// TIA Portal project "Ejercicio2" (V15.1)

(* hardware
DEVICE "S7-1200 station_2"  S7-1200 Station
   slot 0: "Rack_0"  S7-1200 Rack  Rack  V1.0
   slot 1: "PLC_0"  CPU 1215C AC/DC/Rly  6ES7 215-1BG40-0XB0  V4.2
DEVICE "HMI_1"  KTP700 Basic PN Portrait
   slot 0: "HMI_1"  KTP700 Basic PN Portrait  6AV2 123-2GB03-0AX0  15.1.0.0
   slot 1: "HMI_RT_1"  KTP700 Basic PN Portrait  6AV2 123-2GB03-0AX0  15.1.0.0
   slot 5: "HMI_1.IE_CP_1"  PROFINET Interface  15.0.1.0
      slot 1: "Interfaz PROFINET_1"  PROFINET Interface
         slot 1: "Port_1"  Port
*)

// ===== PLC "PLC_0"  CPU 1215C AC/DC/Rly =====

VAR_GLOBAL   // PLC tag table "Tabla de variables estándar"
   "Zona 1" AT %M0.0 : Bool;   // Entrada delantera, sala de estar, cocina y dormitorio 3
   "Zona 2" AT %M0.1 : Bool;   // Dormitorio 1, dormitorio 2, baño y entrada trasera
   "Alarma ON/OFF" AT %M0.2 : Bool;   // Activa o desactiva el sistema de alarma.
   "Alarma manual" AT %M0.3 : Bool;   // Permite activar manualmente la sirena de alarma
   "LED sistema de alarma" AT %M10.0 : Bool;   // Estará encendido si está activado y parpadeante si está desactivado, estando abiertas la zona 1 o la zona 2
   "Sirena de alarma" AT %M10.1 : Bool;   // Dispara la sirena de alarma
   "Señal de alerta baja" AT %M10.2 : Bool;   // Activa una señal de alerta baja que indica que la alarma se disparará al cabo de un número predeterminado de segundos
   "Activar relé" AT %M10.3 : Bool;   // Activa un relé de interface externo (p.ej. para arrancar una marcación automática).
   "Estado Alarma" AT %M1.0 : Bool;   // Usaremos esta variable para detectar cuando el temporizador de 90 segundos haya pasado
   "Estado Sirena" AT %M1.1 : Bool;   // Usaremos esta variable para detectar si alguna zona esta abierta o no
END_VAR

// folder: System blocks/Program resources

DATA_BLOCK "Temporizador 90s"   // DB1
{ S7_Optimized_Access := 'TRUE' }
AUTHOR : Simatic
FAMILY : IEC
NAME : IEC_TMR
VERSION : 1.0
// stored: InstanceOfName IEC_TIMER
"IEC_TIMER"
BEGIN
END_DATA_BLOCK

DATA_BLOCK "Temporizador notificador 60s"   // DB3
{ S7_Optimized_Access := 'TRUE' }
AUTHOR : Simatic
FAMILY : IEC
NAME : IEC_TMR
VERSION : 1.0
// stored: InstanceOfName IEC_TIMER
"IEC_TIMER"
BEGIN
END_DATA_BLOCK

// folder: (top level)

ORGANIZATION_BLOCK "Main"   // OB1, LAD, ProgramCycle
TITLE = "Main Program Sweep (Cycle)"
{ S7_Optimized_Access := 'TRUE' }
VERSION : 0.1
   VAR_INPUT
      Initial_Call : Bool;   // Initial call of this OB
      Remanence : Bool;   // =True, if remanent data are available
   END_VAR
   VAR_TEMP   // added for the SCL form of the ladder/FBD networks
      _w1 : Bool;
   END_VAR
BEGIN

REGION Network 1: Estará encendido si está activado y parpadeante si está desactivado, estando abiertas la zona 1 o la zona 2
   // Si el sistema no está activado, el LED (M10.0) parpadea al estar abiertas la zona 1 (%M0.0) o 2 (%M0.1).
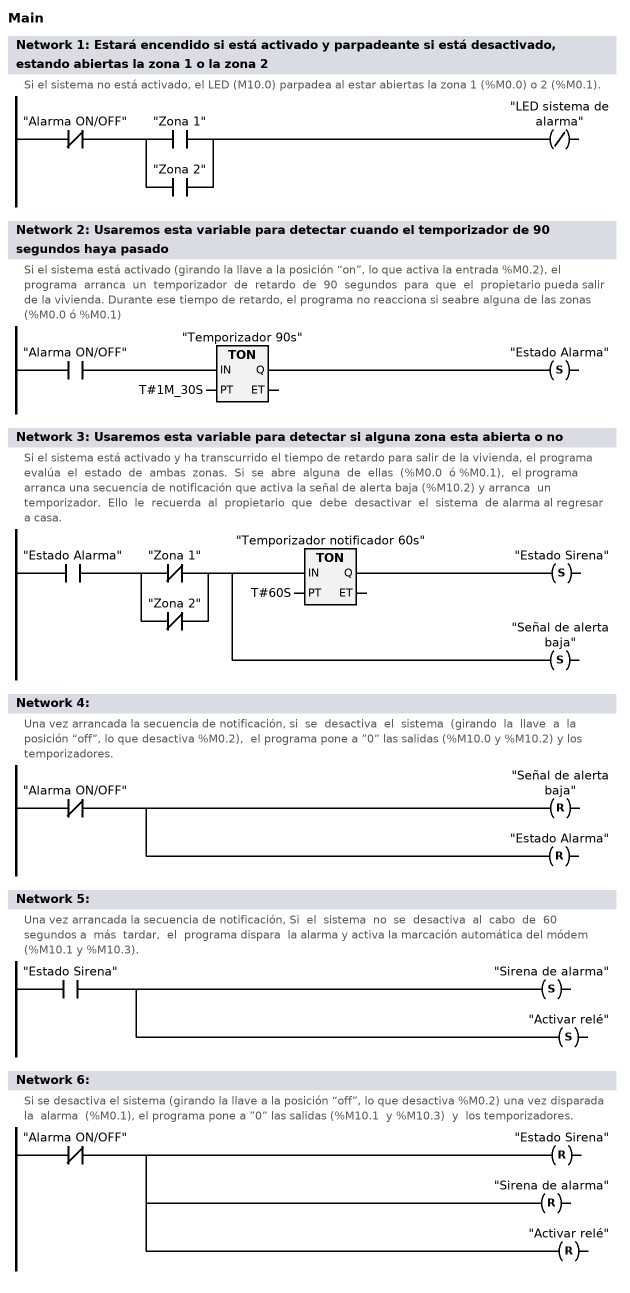
   RUNG wire#powerrail
      I_Contact( "Alarma ON/OFF" )
      wire#w1
      Contact( "Zona 1" )
      wire#w2
      I_Coil( "LED sistema de alarma" )
   END_RUNG
   RUNG wire#w1
      Contact( "Zona 2" )
   END_RUNG wire#w2
   // the same network as SCL:
   "LED sistema de alarma" := NOT (NOT "Alarma ON/OFF" AND ("Zona 1" OR "Zona 2"));
END_REGION

REGION Network 2: Usaremos esta variable para detectar cuando el temporizador de 90 segundos haya pasado
   // Si el sistema está activado (girando la llave a la posición “on”, lo que activa la entrada %M0.2), el  programa  arranca  un  temporizador  de  retardo  de  90  segundos  para  que  el  propietario pueda salir de la vivienda. Durante ese tiempo de retardo, el programa no reacciona si seabre alguna de las zonas (%M0.0 ó %M0.1)
   "Temporizador 90s".TON(IN := "Alarma ON/OFF", PT := T#1M_30S);
   IF "Temporizador 90s".Q THEN "Estado Alarma" := TRUE; END_IF;
END_REGION

REGION Network 3: Usaremos esta variable para detectar si alguna zona esta abierta o no
   // Si el sistema está activado y ha transcurrido el tiempo de retardo para salir de la vivienda, el programa  evalúa  el  estado  de  ambas  zonas.  Si  se  abre  alguna  de  ellas  (%M0.0  ó %M0.1),  el programa arranca una secuencia de notificación que activa la señal de alerta baja (%M10.2) y arranca  un  temporizador.  Ello  le  recuerda  al  propietario  que  debe  desactivar  el  sistema  de alarma al regresar a casa.
   #_w1 := "Estado Alarma" AND (NOT "Zona 1" OR NOT "Zona 2");
   "Temporizador notificador 60s".TON(IN := #_w1, PT := T#60S);
   IF "Temporizador notificador 60s".Q THEN "Estado Sirena" := TRUE; END_IF;
   IF #_w1 THEN "Señal de alerta baja" := TRUE; END_IF;
END_REGION

REGION Network 4
   // Una vez arrancada la secuencia de notificación, si  se  desactiva  el  sistema  (girando  la  llave  a  la  posición “off”, lo que desactiva %M0.2),  el programa pone a ”0” las salidas (%M10.0 y %M10.2) y los temporizadores.
   RUNG wire#powerrail
      I_Contact( "Alarma ON/OFF" )
      wire#w1
      R_Coil( "Señal de alerta baja" )
   END_RUNG
   RUNG wire#w1
      R_Coil( "Estado Alarma" )
   END_RUNG
   // the same network as SCL:
   IF NOT "Alarma ON/OFF" THEN
       "Señal de alerta baja" := FALSE;
       "Estado Alarma" := FALSE;
   END_IF;
END_REGION

REGION Network 5
   // Una vez arrancada la secuencia de notificación, Si  el  sistema  no  se  desactiva  al  cabo  de  60  segundos a  más  tardar,  el  programa dispara  la alarma y activa la marcación automática del módem (%M10.1 y %M10.3).
   RUNG wire#powerrail
      Contact( "Estado Sirena" )
      wire#w1
      S_Coil( "Sirena de alarma" )
   END_RUNG
   RUNG wire#w1
      S_Coil( "Activar relé" )
   END_RUNG
   // the same network as SCL:
   IF "Estado Sirena" THEN
       "Sirena de alarma" := TRUE;
       "Activar relé" := TRUE;
   END_IF;
END_REGION

REGION Network 6
   // Si se desactiva el sistema (girando la llave a la posición “off”, lo que desactiva %M0.2) una vez disparada  la  alarma  (%M0.1), el programa pone a ”0” las salidas (%M10.1  y %M10.3)  y  los temporizadores.
   RUNG wire#powerrail
      I_Contact( "Alarma ON/OFF" )
      wire#w1
      R_Coil( "Estado Sirena" )
   END_RUNG
   RUNG wire#w1
      R_Coil( "Sirena de alarma" )
   END_RUNG
   RUNG wire#w1
      R_Coil( "Activar relé" )
   END_RUNG
   // the same network as SCL:
   IF NOT "Alarma ON/OFF" THEN
       "Estado Sirena" := FALSE;
       "Sirena de alarma" := FALSE;
       "Activar relé" := FALSE;
   END_IF;
END_REGION
END_ORGANIZATION_BLOCK

(* ===== HMI "HMI_RT_1" =====
system functions are stored by id; their names below are inferred from use
connection "HMI_Conexión_1": ETHERNET, SMART_S7_1200_OMS

HMI tags "Tabla de variables estándar"
   "Número_imagen_variable" : UInt, internal
   "Alarma ON/OFF" : Bool = PLC "Alarma ON/OFF" AT %M0.2, 1 s
   "LED sistema de alarma" : Bool = PLC "LED sistema de alarma" AT %M10.0, 1 s
   "Señal de alerta baja" : Bool = PLC "Señal de alerta baja" AT %M10.2, 1 s
   "Sirena de alarma" : Bool = PLC "Sirena de alarma" AT %M10.1, 1 s
   "Activar relé" : Bool = PLC "Activar relé" AT %M10.3, 1 s

text list "Nombre_imagen_lista_texto": 1 'Imagen raíz'

Template "Plantilla_1" 480x800
   Button "Template_Button" at 428,727 size 50x71; TextOff 'Text'
   Button "Template_Button_1" at 375,727 size 50x71; TextOff 'Text'
   Button "Template_Button_2" at 321,727 size 50x71; TextOff 'Text'
   Button "Template_Button_3" at 268,727 size 50x71; TextOff 'Text'
   Button "Template_Button_4" at 214,727 size 50x71; TextOff 'Text'
   Button "Template_Button_5" at 161,727 size 50x71; TextOff 'Text'
   Button "Template_Button_6" at 108,727 size 50x71; TextOff 'Text'
   Button "Template_Button_7" at 54,727 size 50x71; TextOff 'Text'
   Button "Avisos" at 1,727 size 50x71; TextOff 'Avisos'; PictureOff "AlarmDisplay_KTP700_Basic_PN_Portrait_TR"; PictureOn "AlarmDisplay_KTP700_Basic_PN_Portrait_TR"
      on Release: function_ef3f5d25("Ventana de avisos_no_acusado", -1)
   SymbolicIOField "Imagen_campo_ES_simbólico" at 2,11 size 371x38; TextOff '0'; TextOn '1'; TextList "Nombre_imagen_lista_texto"
      ProcessValue <- "Número_imagen_variable"
      on Change: ActivateScreenByNumber("Número_imagen_variable", 0)
   DateTimeField "HmiScreenItemData" at 375,30 size 105x30
   DateTimeField "HmiScreenItemData_1" at 375,0 size 105x30

screen "Imagen raíz" 480x800, template "Plantilla_1"
   on GenerateScreen: SetTag("Número_imagen_variable", 1)
   TextField "Campo de texto_1" at 21,75 size 127x23; Text 'Activar Alarma'
   Switch "Interruptor_1" at 56,109 size 64x32; CaptionText 'Switch'; TextOff 'OFF'; TextOn 'ON'
      ProcessValue <- "Alarma ON/OFF"
   Circle "Círculo_1" at 333,109 size 48x48
      Appearance <- "LED sistema de alarma"
   TextField "Campo de texto_2" at 274,76 size 158x23; Text 'LED estado alarma'
   Circle "Círculo_2" at 157,213 size 48x48
      Appearance <- "Señal de alerta baja"
   TextField "Campo de texto_3" at 213,227 size 141x23; Text 'Estado de Alerta'
   Circle "Círculo_3" at 158,307 size 48x48
      Appearance <- "Sirena de alarma"
   TextField "Campo de texto_4" at 218,319 size 57x23; Text 'Sirena'
   Circle "Círculo_4" at 157,360 size 48x48
      Appearance <- "Activar relé"
   TextField "Campo de texto_5" at 218,372 size 178x23; Text 'Aviso a policía (Relé)'
*)